PROGRAM Group_08_Logic
VAR
	TON_0: TON;
	TON_1: TON;
	TON_2: TON;
	TON_3: TON;
	
Axis_24_Velocity_Range: LREAL;
Axis_24_Velocity_Scale: LREAL;
Axis_24_Velocity_Raw: LREAL;
Axis_24_Soft_Range: LREAL;
Axis_24_Soft_Position: LREAL;
Axis_24_Soft_Position_In_Range: LREAL;
END_VAR
VAR // added by the converter: edge detectors and wires of the graphical bodies
    _w1, _w2, _w3, _w4, _w5, _w6, _w7, _w8, _w9, _w10, _w11, _w12, _w13, _w14, _w15, _w16, _w17, _w18, _w19, _w20, _w21, _w22, _w23, _w24, _w25, _w26, _w27, _w28, _w29, _w30, _w31, _w32 : BOOL;
END_VAR

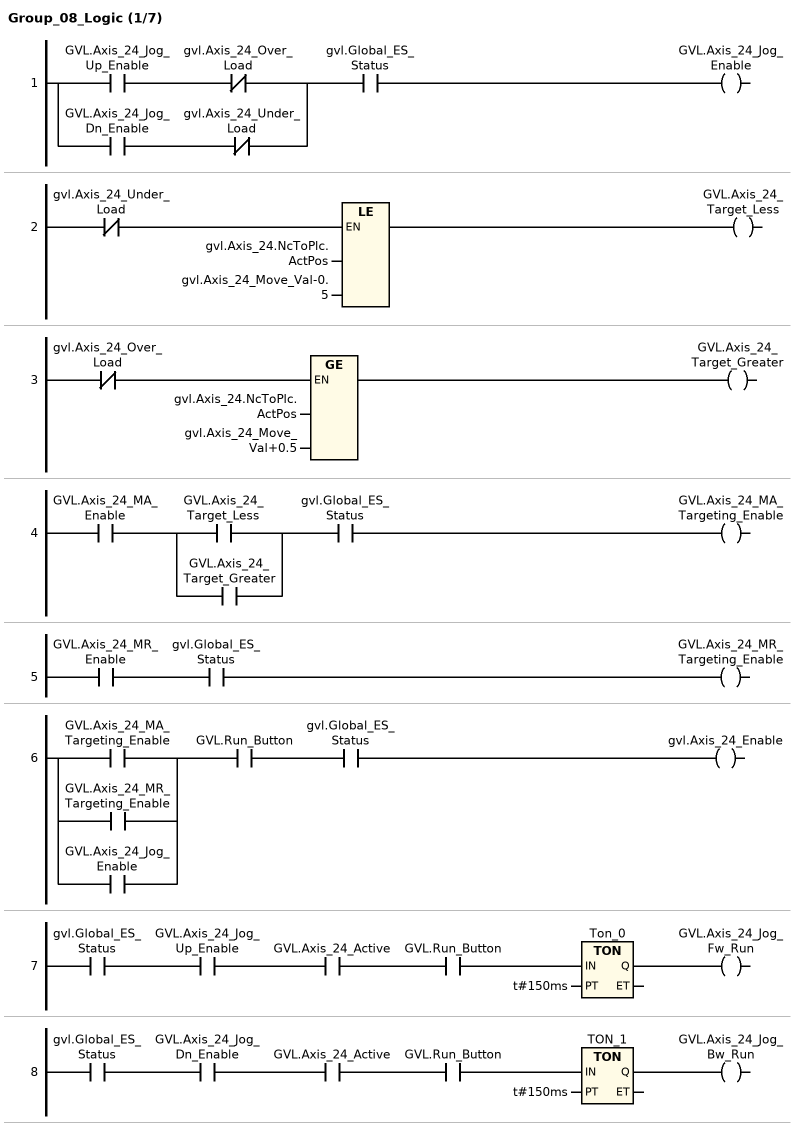
// NETWORK 1
GVL.Axis_24_Jog_Enable := (GVL.Axis_24_Jog_Up_Enable AND NOT gvl.Axis_24_Over_Load OR GVL.Axis_24_Jog_Dn_Enable AND NOT gvl.Axis_24_Under_Load) AND gvl.Global_ES_Status;

// NETWORK 2
GVL.Axis_24_Target_Less := NOT gvl.Axis_24_Under_Load AND gvl.Axis_24.NcToPlc.ActPos <= (gvl.Axis_24_Move_Val-0.5);

// NETWORK 3
GVL.Axis_24_Target_Greater := NOT gvl.Axis_24_Over_Load AND gvl.Axis_24.NcToPlc.ActPos >= (gvl.Axis_24_Move_Val+0.5);

// NETWORK 4
GVL.Axis_24_MA_Targeting_Enable := GVL.Axis_24_MA_Enable AND (GVL.Axis_24_Target_Less OR GVL.Axis_24_Target_Greater) AND gvl.Global_ES_Status;

// NETWORK 5
GVL.Axis_24_MR_Targeting_Enable := GVL.Axis_24_MR_Enable AND gvl.Global_ES_Status;

// NETWORK 6
gvl.Axis_24_Enable := (GVL.Axis_24_MA_Targeting_Enable OR GVL.Axis_24_MR_Targeting_Enable OR GVL.Axis_24_Jog_Enable) AND GVL.Run_Button AND gvl.Global_ES_Status;

// NETWORK 7
Ton_0(IN := gvl.Global_ES_Status AND GVL.Axis_24_Jog_Up_Enable AND GVL.Axis_24_Active AND GVL.Run_Button, PT := t#150ms); // TON
GVL.Axis_24_Jog_Fw_Run := Ton_0.Q;

// NETWORK 8
TON_1(IN := gvl.Global_ES_Status AND GVL.Axis_24_Jog_Dn_Enable AND GVL.Axis_24_Active AND GVL.Run_Button, PT := t#150ms); // TON
GVL.Axis_24_Jog_Bw_Run := TON_1.Q;

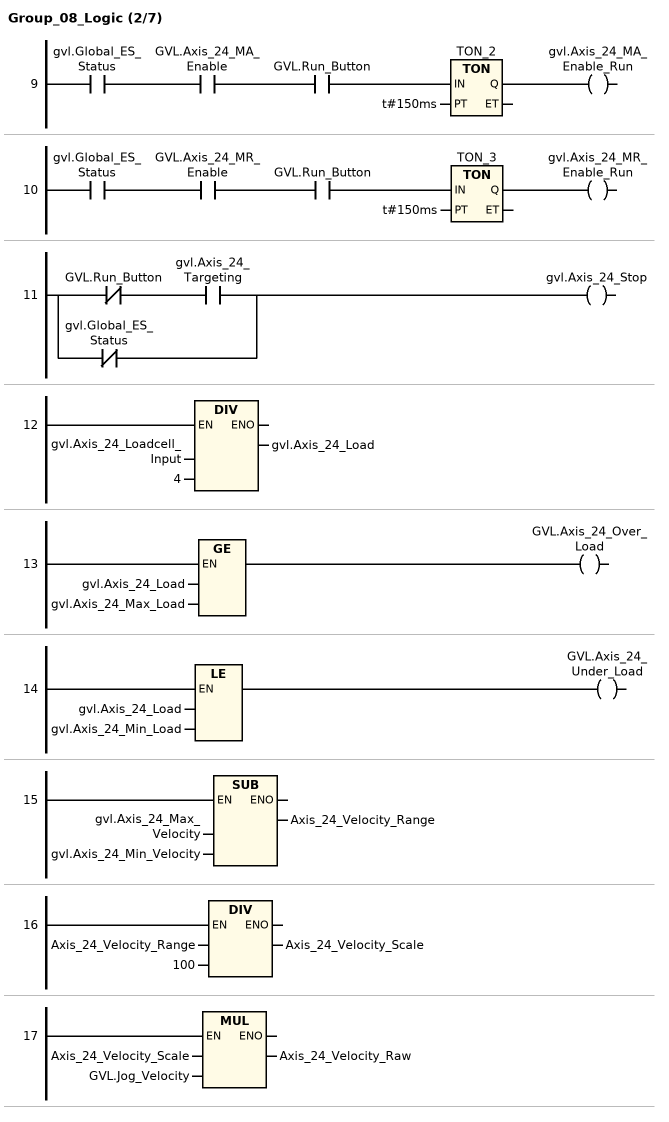
// NETWORK 9
TON_2(IN := gvl.Global_ES_Status AND GVL.Axis_24_MA_Enable AND GVL.Run_Button, PT := t#150ms); // TON
gvl.Axis_24_MA_Enable_Run := TON_2.Q;

// NETWORK 10
TON_3(IN := gvl.Global_ES_Status AND GVL.Axis_24_MR_Enable AND GVL.Run_Button, PT := t#150ms); // TON
gvl.Axis_24_MR_Enable_Run := TON_3.Q;

// NETWORK 11
gvl.Axis_24_Stop := NOT GVL.Run_Button AND gvl.Axis_24_Targeting OR NOT gvl.Global_ES_Status;

// NETWORK 12
gvl.Axis_24_Load := gvl.Axis_24_Loadcell_Input / 4;

// NETWORK 13
GVL.Axis_24_Over_Load := gvl.Axis_24_Load >= gvl.Axis_24_Max_Load;

// NETWORK 14
GVL.Axis_24_Under_Load := gvl.Axis_24_Load <= gvl.Axis_24_Min_Load;

// NETWORK 15
Axis_24_Velocity_Range := gvl.Axis_24_Max_Velocity - gvl.Axis_24_Min_Velocity;

// NETWORK 16
Axis_24_Velocity_Scale := Axis_24_Velocity_Range / 100;

// NETWORK 17
Axis_24_Velocity_Raw := Axis_24_Velocity_Scale * GVL.Jog_Velocity;

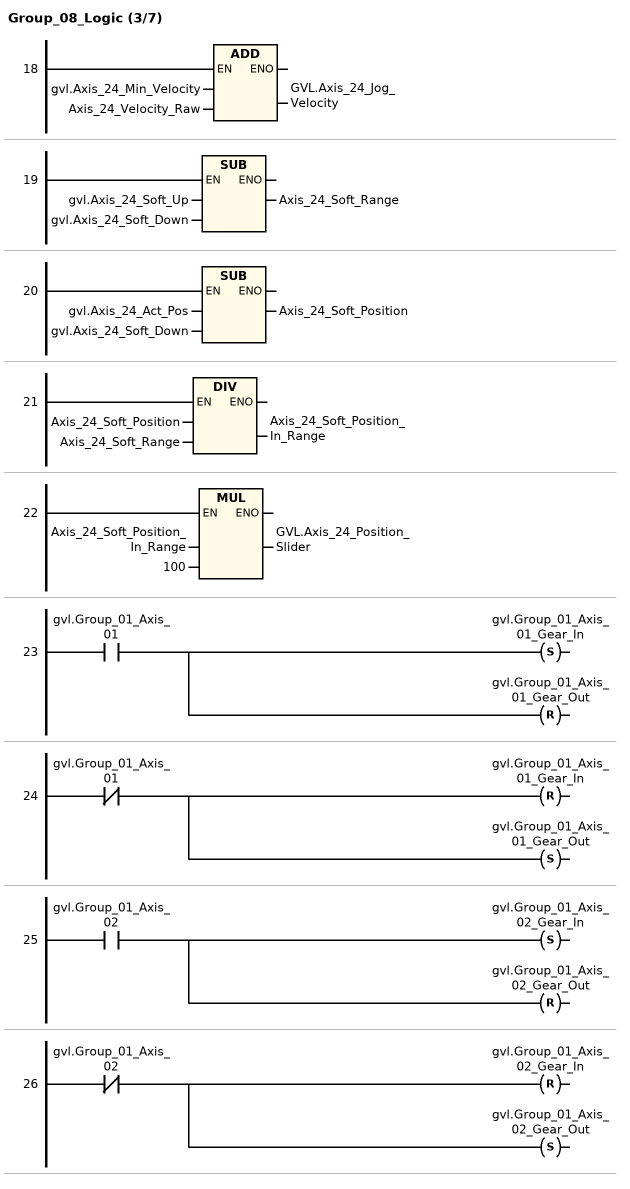
// NETWORK 18
GVL.Axis_24_Jog_Velocity := gvl.Axis_24_Min_Velocity + Axis_24_Velocity_Raw;

// NETWORK 19
Axis_24_Soft_Range := gvl.Axis_24_Soft_Up - gvl.Axis_24_Soft_Down;

// NETWORK 20
Axis_24_Soft_Position := gvl.Axis_24_Act_Pos - gvl.Axis_24_Soft_Down;

// NETWORK 21
Axis_24_Soft_Position_In_Range := Axis_24_Soft_Position / Axis_24_Soft_Range;

// NETWORK 22
GVL.Axis_24_Position_Slider := Axis_24_Soft_Position_In_Range * 100;

// NETWORK 23
_w1 := gvl.Group_01_Axis_01;
gvl.Group_01_Axis_01_Gear_In S= _w1;
gvl.Group_01_Axis_01_Gear_Out R= _w1;

// NETWORK 24
_w2 := NOT gvl.Group_01_Axis_01;
gvl.Group_01_Axis_01_Gear_In R= _w2;
gvl.Group_01_Axis_01_Gear_Out S= _w2;

// NETWORK 25
_w3 := gvl.Group_01_Axis_02;
gvl.Group_01_Axis_02_Gear_In S= _w3;
gvl.Group_01_Axis_02_Gear_Out R= _w3;

// NETWORK 26
_w4 := NOT gvl.Group_01_Axis_02;
gvl.Group_01_Axis_02_Gear_In R= _w4;
gvl.Group_01_Axis_02_Gear_Out S= _w4;

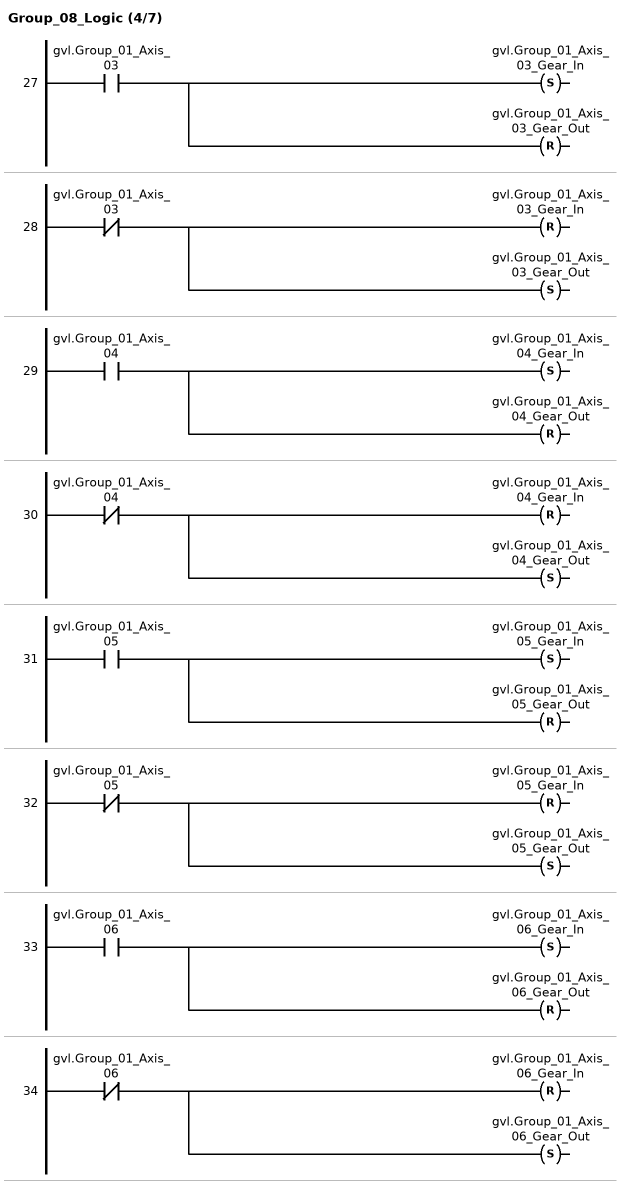
// NETWORK 27
_w5 := gvl.Group_01_Axis_03;
gvl.Group_01_Axis_03_Gear_In S= _w5;
gvl.Group_01_Axis_03_Gear_Out R= _w5;

// NETWORK 28
_w6 := NOT gvl.Group_01_Axis_03;
gvl.Group_01_Axis_03_Gear_In R= _w6;
gvl.Group_01_Axis_03_Gear_Out S= _w6;

// NETWORK 29
_w7 := gvl.Group_01_Axis_04;
gvl.Group_01_Axis_04_Gear_In S= _w7;
gvl.Group_01_Axis_04_Gear_Out R= _w7;

// NETWORK 30
_w8 := NOT gvl.Group_01_Axis_04;
gvl.Group_01_Axis_04_Gear_In R= _w8;
gvl.Group_01_Axis_04_Gear_Out S= _w8;

// NETWORK 31
_w9 := gvl.Group_01_Axis_05;
gvl.Group_01_Axis_05_Gear_In S= _w9;
gvl.Group_01_Axis_05_Gear_Out R= _w9;

// NETWORK 32
_w10 := NOT gvl.Group_01_Axis_05;
gvl.Group_01_Axis_05_Gear_In R= _w10;
gvl.Group_01_Axis_05_Gear_Out S= _w10;

// NETWORK 33
_w11 := gvl.Group_01_Axis_06;
gvl.Group_01_Axis_06_Gear_In S= _w11;
gvl.Group_01_Axis_06_Gear_Out R= _w11;

// NETWORK 34
_w12 := NOT gvl.Group_01_Axis_06;
gvl.Group_01_Axis_06_Gear_In R= _w12;
gvl.Group_01_Axis_06_Gear_Out S= _w12;

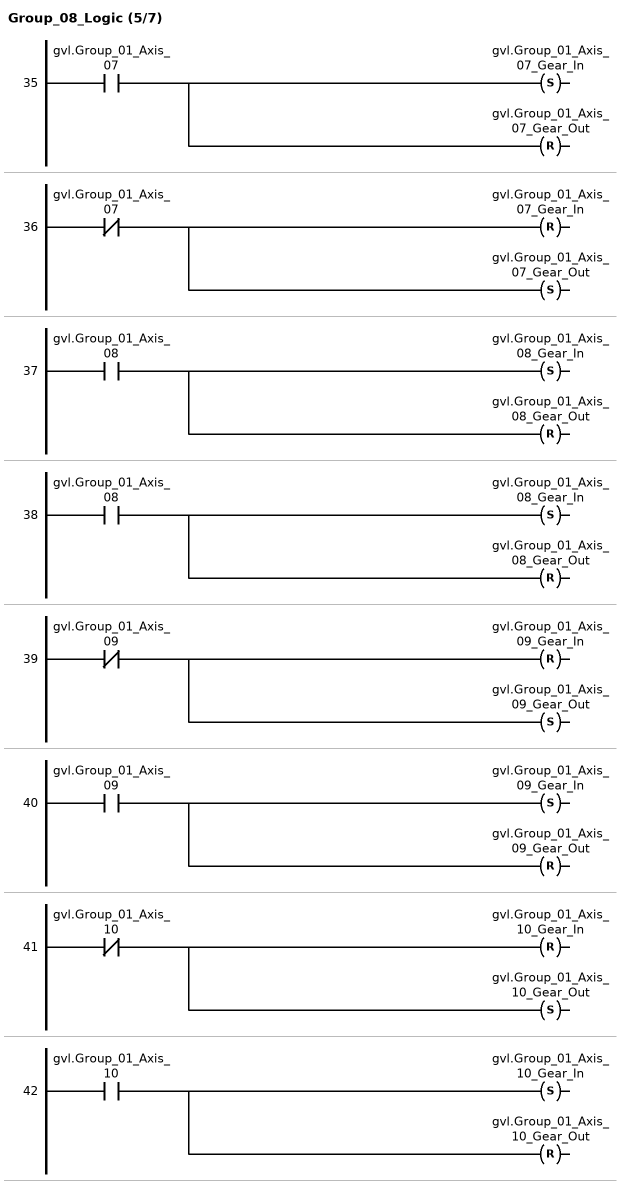
// NETWORK 35
_w13 := gvl.Group_01_Axis_07;
gvl.Group_01_Axis_07_Gear_In S= _w13;
gvl.Group_01_Axis_07_Gear_Out R= _w13;

// NETWORK 36
_w14 := NOT gvl.Group_01_Axis_07;
gvl.Group_01_Axis_07_Gear_In R= _w14;
gvl.Group_01_Axis_07_Gear_Out S= _w14;

// NETWORK 37
_w15 := gvl.Group_01_Axis_08;
gvl.Group_01_Axis_08_Gear_In S= _w15;
gvl.Group_01_Axis_08_Gear_Out R= _w15;

// NETWORK 38
_w16 := gvl.Group_01_Axis_08;
gvl.Group_01_Axis_08_Gear_In S= _w16;
gvl.Group_01_Axis_08_Gear_Out R= _w16;

// NETWORK 39
_w17 := NOT gvl.Group_01_Axis_09;
gvl.Group_01_Axis_09_Gear_In R= _w17;
gvl.Group_01_Axis_09_Gear_Out S= _w17;

// NETWORK 40
_w18 := gvl.Group_01_Axis_09;
gvl.Group_01_Axis_09_Gear_In S= _w18;
gvl.Group_01_Axis_09_Gear_Out R= _w18;

// NETWORK 41
_w19 := NOT gvl.Group_01_Axis_10;
gvl.Group_01_Axis_10_Gear_In R= _w19;
gvl.Group_01_Axis_10_Gear_Out S= _w19;

// NETWORK 42
_w20 := gvl.Group_01_Axis_10;
gvl.Group_01_Axis_10_Gear_In S= _w20;
gvl.Group_01_Axis_10_Gear_Out R= _w20;

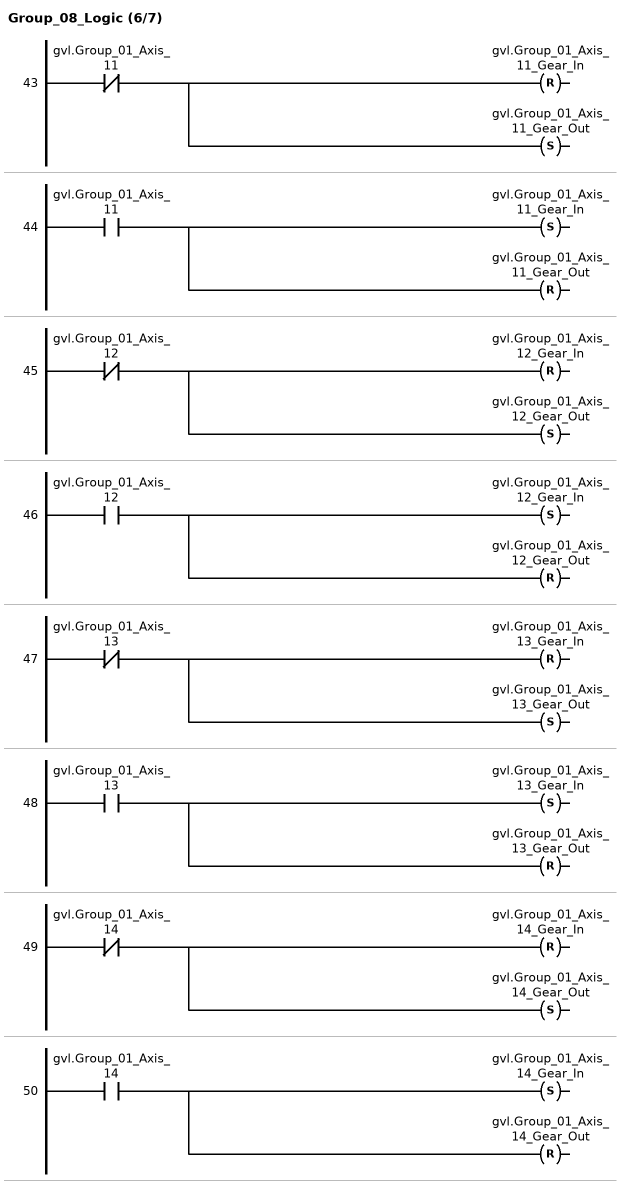
// NETWORK 43
_w21 := NOT gvl.Group_01_Axis_11;
gvl.Group_01_Axis_11_Gear_In R= _w21;
gvl.Group_01_Axis_11_Gear_Out S= _w21;

// NETWORK 44
_w22 := gvl.Group_01_Axis_11;
gvl.Group_01_Axis_11_Gear_In S= _w22;
gvl.Group_01_Axis_11_Gear_Out R= _w22;

// NETWORK 45
_w23 := NOT gvl.Group_01_Axis_12;
gvl.Group_01_Axis_12_Gear_In R= _w23;
gvl.Group_01_Axis_12_Gear_Out S= _w23;

// NETWORK 46
_w24 := gvl.Group_01_Axis_12;
gvl.Group_01_Axis_12_Gear_In S= _w24;
gvl.Group_01_Axis_12_Gear_Out R= _w24;

// NETWORK 47
_w25 := NOT gvl.Group_01_Axis_13;
gvl.Group_01_Axis_13_Gear_In R= _w25;
gvl.Group_01_Axis_13_Gear_Out S= _w25;

// NETWORK 48
_w26 := gvl.Group_01_Axis_13;
gvl.Group_01_Axis_13_Gear_In S= _w26;
gvl.Group_01_Axis_13_Gear_Out R= _w26;

// NETWORK 49
_w27 := NOT gvl.Group_01_Axis_14;
gvl.Group_01_Axis_14_Gear_In R= _w27;
gvl.Group_01_Axis_14_Gear_Out S= _w27;

// NETWORK 50
_w28 := gvl.Group_01_Axis_14;
gvl.Group_01_Axis_14_Gear_In S= _w28;
gvl.Group_01_Axis_14_Gear_Out R= _w28;

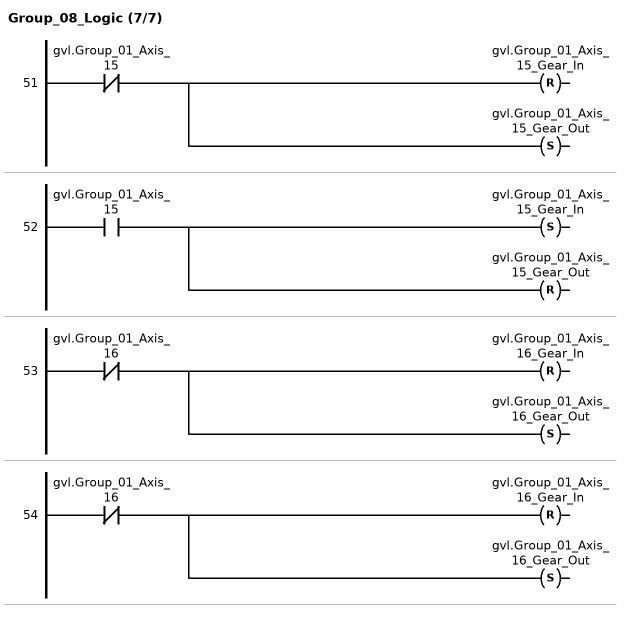
// NETWORK 51
_w29 := NOT gvl.Group_01_Axis_15;
gvl.Group_01_Axis_15_Gear_In R= _w29;
gvl.Group_01_Axis_15_Gear_Out S= _w29;

// NETWORK 52
_w30 := gvl.Group_01_Axis_15;
gvl.Group_01_Axis_15_Gear_In S= _w30;
gvl.Group_01_Axis_15_Gear_Out R= _w30;

// NETWORK 53
_w31 := NOT gvl.Group_01_Axis_16;
gvl.Group_01_Axis_16_Gear_In R= _w31;
gvl.Group_01_Axis_16_Gear_Out S= _w31;

// NETWORK 54
_w32 := NOT gvl.Group_01_Axis_16;
gvl.Group_01_Axis_16_Gear_In R= _w32;
gvl.Group_01_Axis_16_Gear_Out S= _w32;

END_PROGRAM

(* stored: Version 1.1.0.1, ProductVersion 3.1.4022.12
   POU Group_08_Logic: Id {9e963177-3830-4326-b910-f129e6859622}, SpecialFunc None *)
